FUNCTION Convert_UINT_TO_WORD : Hresult
VAR_INPUT
	in : UINT;
	out : REFERENCE TO WORD;
END_VAR
VAR
	converted : WORD;
END_VAR
VAR CONSTANT
	INCOMPATIBLE : HRESULT := 16#9811070E;
END_VAR

converted := UINT_TO_WORD(in);

IF (WORD_TO_UINT(converted) <> in) THEN
	Convert_UINT_TO_WORD := INCOMPATIBLE;
	RETURN;
END_IF

out := converted;

END_FUNCTION

(* stored: Version 1.1.0.1, ProductVersion 3.1.4024.12
   POU Convert_UINT_TO_WORD: Id {e1d704d3-a22b-4b9b-a9f7-c6936ebf0868}, SpecialFunc None *)
